ABB RAPID module: MainModule.mod

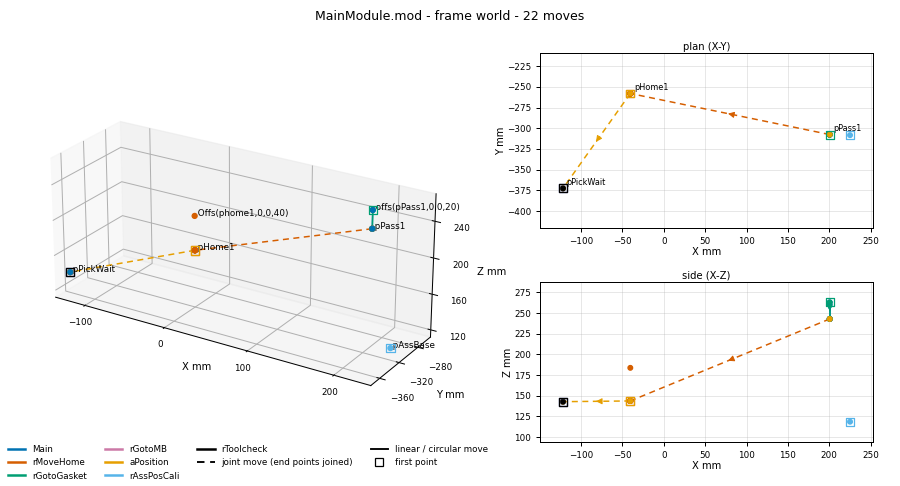
[picture p0: tool path of MainModule.mod in frame world, 22 of 155 moves have a stored position in this frame; points joined in program order, loops and branches not executed]
 MODULE MainModule
!*****************************************************
!Module Name: MainModule
!Version:     2.0
!Description: Menu Buttun and Gasket Assembly station
!Date:        2014\04\28
!Author:      Gavin Zhang
!*****************************************************
     PROC Main()
        VAR num X;
        VAR num Y;
        VAR string str_i;
        VAR pose poseCCD1;
        VAR pose poseTool;
        VAR num anglex;
        VAR num angley;
        VAR num anglez;
        rInitall;
        WHILE TRUE DO
            WHILE SocketStr<>"" DO
                IF SocketStr="robottest" THEN
                    FOR i FROM 1 TO 100 DO
                        SockGet:=FALSE;
                        MoveJ pPickWait,v200,z50,tGripper;
                        MoveL pCCD1,v200,fine,tGripper;
                        WaitTime 0.5;
                        SendStr:="ok";
                        SocketStr:="";
                        WaitUntil SendStr="";
                        waittime 0.5;
                        SockGet:=TRUE;
                        WaitUntil SocketStr="ok,ccd1check";
                        SocketStr:="";
                    ENDFOR
                    SockGet:=TRUE;
                ELSEIF SocketStr="robottest2" THEN
                    FOR i FROM 1 TO 50 DO
                        SockGet:=FALSE;
                        MoveL offs(pCCD1,0,0,20),v200,fine,tGripper;
                        MoveL pCCD1,v200,fine,tGripper;
                        MoveL offs(pCCD1,0,0,20),v200,fine,tGripper;
                        MoveJ offs(pPass1,0,0,20),v300,z10,tGripper;
                        MoveL pPass1,v600,z10,tGripper;
                        AccSet 50,50;
                        !MoveJ pInsert,v300,fine,tCurtool\WObj:=AssFrame;
                        MoveL pInsert,v300,fine,tCurtool\WObj:=AssFrame;
                        rInsert1;
                        WaitTime 0.5;
                        pActPos:=CRobT(\Tool:=tGripper\wobj:=wobj0);
                        MoveL offs(pActPos,0,0,20),v300,fine,tGripper\WObj:=wobj0;
                        MoveL offs(pCCD1,0,0,20),v200,fine,tGripper;
                        MoveL pCCD1,v200,fine,tGripper;
                        WaitTime 0.5;
                        SendStr:="ok";
                        SocketStr:="";
                        WaitUntil SendStr="";
                        waittime 0.5;
                        SockGet:=TRUE;
                        WaitUntil SocketStr="ok,ccd1check";
                        SocketStr:="";
                    ENDFOR
                    SockGet:=TRUE;
                ELSEIF SocketStr="ccd1check" THEN
                    SockGet:=FALSE;
                    !pCCD1Cali:=pCCD1;
                    MoveL pCCD1Cali,v100,fine,tGripper;
                    WaitTime\InPos,1;
                    SendStr:="ok,ccd1";
                    SocketStr:="";
                    WaitUntil SendStr="";
                    SockGet:=TRUE;
                    WaitUntil SocketStr="ok,ccd1";
                    SockGet:=FALSE;
                    pActPos:=CRobT(\Tool:=tGripper\wobj:=wobj0);
                    SendStr:="ok,"+ValToStr(pActPos.trans.X)+","+ValToStr(pActPos.trans.Y);
                    WaitUntil SendStr="";
                    SocketStr:="";
                    SockGet:=TRUE;
                    WaitUntil SocketStr="ccd1checkfinish";
                    SocketStr:="";
                    MoveJ pHome1,v100,fine,tGripper;
                    MoveJ pHome,v100,fine,tGripper;
                ELSEIF SocketStr="ccd2check" THEN
                    SockGet:=FALSE;
                    MoveJ phome,v100,z5,tGripper;
                    !MoveJ offs(pCCD2Cali,0,0,30),v100,z5,tGripper;
                    FOR i FROM 1 TO 9 DO
                        n:=trunc((i-1)/3);
                        b:=i-n*3;
                        pccd2Calib_T{i}:=offs(pCCD2Cali,(n-1)*2,(b-2)*2,0);
                    ENDFOR
                    FOR i FROM 1 TO 9 DO
                        MoveJ offs(pPickInkpad,0,0,140),v300,z5,tGripper;
                        MoveL pPickInkpad,v100,fine,tGripper;
                        WaitTime 0.5;
                        MoveL offs(pPickInkpad,0,0,140),v300,z5,tGripper;
                        SockGet:=FALSE;
                        MoveL offs(pccd2Calib_T{ARRAY{i}},0,0,30),v300,fine,tGripper;
                        MoveL pccd2Calib_T{ARRAY{i}},v100,fine,tGripper;
                        WaitTime\InPos,1;
                        pActPos:=CRobT(\Tool:=tGripper\wobj:=wobj0);
                        nPOSCCD2{i}:=pActPos.trans;
                        CCD2X{i}:=ValToStr(pActPos.trans.x);
                        CCD2y{i}:=ValToStr(pActPos.trans.y);
                        str_i:=ValToStr(i);
                        SendStr:="ok,"+str_i+","+CCD2X{i}+","+CCD2y{i};
                        WaitUntil SendStr="";
                        SocketStr:="";
                        SockGet:=TRUE;
                        IF i<>9 THEN
                            WaitUntil SocketStr="ok,ccd2";
                        ENDIF
                        WaitTime 1;
                        MoveL offs(pccd2Calib_T{ARRAY{i}},0,0,30),v300,fine,tGripper;
                    ENDFOR
                    SocketStr:="";
                    SockGet:=TRUE;
                    MoveJ phome,v100,z5,tGripper;
                ELSEIF SocketStr="gotomenubnt" THEN
                    SockGet:=FALSE;
                    rMoveHome;
                    MoveL pPickWait,v1000,fine,tGripper;
                    MoveL offs(pPick,0,0,30),v400,fine,tGripper;
                    MoveL pPick,v100,fine,tGripper;
                    SendStr:="ok";
                    SocketStr:="";
                    WaitUntil SendStr="";
                    SockGet:=TRUE;
                    !MoveL offs(pPick,0,0,30),v400,fine,tGripper;
                ELSEIF SocketStr="gotombccd" THEN
                    SockGet:=FALSE;
                    MoveL offs(pPick,0,0,30),v50,fine,tGripper;
                    !rMoveHome;
                    MoveL pCCD1,v600,fine,tGripper;
                    SendStr:="ok";
                    WaitTime 0.2;
                    SocketStr:="";
                    WaitUntil SendStr="";
                    SockGet:=TRUE;
                ELSEIF SocketStr="gotogasket" THEN
                    SockGet:=FALSE;
                    rMoveHome;
                    MoveJ pPass1,v600,z10,tCurTool;
                    MoveJ pInsert,v300,fine,tCurtool\WObj:=AssFrame;
                    !SocketSend socket1 \Str:="gotogasketfinish";
                    SendStr:="ok";
                    SocketStr:="";
                    WaitUntil SendStr="";
                    SockGet:=TRUE;
                ELSEIF SocketStr="gotoinitpos" THEN
                    SockGet:=FALSE;
                    rMoveHome;
                    !MoveJ pPass1,v600,z10,tGripper;
                    MoveJ pHome,v600,fine,tGripper;
                    SendStr:="ok";
                    SocketStr:="";
                    WaitUntil SendStr="";
                    SockGet:=TRUE;
                ELSEIF SocketStr="error" THEN
                    SockGet:=FALSE;
                    rMoveHome;
                    SendStr:="ok";
                    SocketStr:="";
                    WaitUntil SendStr="";
                    SockGet:=TRUE;
                ELSEIF SocketStr="startpress" THEN
                    SockGet:=FALSE;
                    rMoveHome;
                    MoveJ pPass1,v600,z10,tGripper;
                    rInsert1;
                    SendStr:="ok";
                    SocketStr:="";
                    WaitUntil SendStr="";
                    SockGet:=TRUE;
                ELSEIF SocketStr="calibtool" THEN
                    rTCPCalib1;
                ELSEIF SocketStr="ccd1calibration" THEN
                    rCCD1Calibration_1;
                ELSEIF SocketStr="calibtool5" THEN
                    rToolcheck;
                ELSEIF SocketStr="ccd2calibration" THEN
                    rCCD2Calibration;
                ELSEIF SocketStr="startwork" THEN
                    rWorkFlow;
                ELSEIF StrPart(SocketStr,1,15)="UpdateRobotData" THEN
                    tJogbycp;
                ENDIF
                rCyclecheck;
            ENDWHILE
            WaitTime 0.2;
        ENDWHILE
    ENDPROC

    PROC rInitall()
        WHILE diCalibration=1 DO
            TPErase;
            TPWrite "The Safe_Door is Opened,Please Close it";
            WaitDI diCalibration,0;
        ENDWHILE
        StartMove;
        AccSet 5,5;
        rMoveHome;
        bEmptyDone:=FALSE;
        SockGet:=TRUE;
        SocketStr:="";
        Reset doRobError1;
        Reset doRobError2;
        Reset doRobError3;
        Reset doRobError4;
        Reset doSocketError;
        Set doReady1;
        IDelete iInitall;
        CONNECT iInitall WITH tInitiall;
        ISignalDI diRobReset,1,iInitall;
        IDelete iInitall;
        CONNECT iInitall WITH tInitiall;
        ISignalDI diHomePos,1,iInitall;
        IDelete iSocketError;
        CONNECT iSocketError WITH tSocketerror;
        ISignalDO doSocketError,1,iSocketError;
        IDelete iEmptydone;
        CONNECT iEmptydone WITH tEmptyDone;
        ISignalDI diEmptydone,1,iEmptydone;
        IDelete intDoor;
        CONNECT intDoor WITH tSafetyDoor;
        ISignalDI diCalibration,1,intDoor;
    ENDPROC

    !rWorkFlow:the robot normal working flow;

    PROC rWorkFlow()
        VAR string str_i;
        !MoveJ pHome,v1000,fine,tGripper;
        WaitUntil SocketStr="startwork";
        SockGet:=FALSE;
        rGotoMB;
        SockGet:=TRUE;
        WaitUntil SocketStr="gotombccd";
        SockGet:=FALSE;
        rGotoMBCCD;
        SockGet:=TRUE;
        WaitUntil SocketStr<>"";
        WaitUntil StrPart(SocketStr,1,10)="workoffset";
        !Stop;
        SockGet:=FALSE;
        rDataOffset;
        SockGet:=TRUE;
        WaitUntil SocketStr<>"";
        WaitUntil StrPart(SocketStr,1,12)="robot_ponits";
        !Stop;
        SockGet:=FALSE;
        rCCD12Offset;
        SockGet:=TRUE;
        WaitUntil SocketStr="gotogasket";
        SockGet:=FALSE;
        rGotoGasket;
        SockGet:=TRUE;
        WaitUntil SocketStr<>"";
        WaitUntil StrPart(SocketStr,1,5)="guide";
        SockGet:=FALSE;
        rCCD3Guide;
        SockGet:=TRUE;
        WaitUntil SocketStr="startpress";
        SockGet:=FALSE;
        rMBPress;
        SockGet:=TRUE;
        WaitTime 0.5;
        !WaitUntil SocketStr= "gotoinitpos";
        SockGet:=FALSE;
        rGotoHome;
        SockGet:=TRUE;
    ENDPROC

    PROC rCyclecheck()
        WaitTime 0.1;
        !SocketStr:="";
    ENDPROC

    PROC rMoveHome()
        VelSet 100,500;
        IF bCurPos(pHome1,tGripper,10,10,10,wobj0) THEN
            MoveJ pHome1,v500,fine,tGripper;
            MoveL pHome,v500,fine,tGripper;
        ENDIF
        IF bCurPos(pHome,tGripper,10,10,10,wobj0) THEN
            MoveL pHome,v500,fine,tGripper;
        ENDIF
        IF bCurPos(pPick,tGripper,10,10,10,wobj0) THEN
            MoveJ offs(pPick,0,0,20),v500,fine,tGripper;
            MoveJ pHome,v500,fine,tGripper;
        ENDIF
        IF bCurPos(pCCD1Cali,tGripper,10,10,10,wobj0) THEN
            !MoveJ pPass1, v500, fine, tGripper;
            MoveJ pHome1,v500,Z10,tGripper;
            MoveL pHome,v500,fine,tGripper;
        ENDIF
        IF bCurPos(pCCD2Cali,tGripper,30,30,10,wobj0) THEN
            MoveJ Offs(pCCD2Cali,0,0,30),v100,fine,tGripper;
            MoveL Offs(phome1,0,0,40),v500,fine,tGripper;
            MoveL pHome,v500,fine,tGripper;
        ENDIF
        IF bCurPos(ppass1,tGripper,10,10,10,wobj0) THEN
            MoveJ pHome1,v500,Z10,tGripper;
            MoveJ pHome,v500,fine,tGripper;
        ENDIF
        IF bCurPos(pInsert,tCurTool,10,10,10,AssFrame) THEN
            MoveJ pPass1,v500,fine,tGripper;
            MoveJ pHome1,v500,fine,tGripper;
            MoveJ pHome,v500,fine,tGripper;
        ENDIF
        IF bCurrentPos(pHome,tGripper)=FALSE THEN
            ! If no known position is found, check if the robot is in a specified
            ! window and move him to the first position in the program
            pActPos:=CRobT(\Tool:=tGripper\WObj:=wobj0);
            IF (pPick.trans.x-5<pActPos.trans.x AND pActPos.trans.x<pCCD2Cali.trans.x+10) AND (-370<pActPos.trans.Y AND pActPos.trans.Y<0) AND pActPos.trans.z>pCCD2Cali.trans.z+20 THEN
                MoveL offs(pActPos,0,0,60),v300,z20,tGripper;
                MoveJ pHome1,v500,fine,tGripper;
                MoveL pHome,v500,fine,tGripper;
            ELSE
                WHILE OpMode()<>OP_MAN_PROG DO
                    TPErase;
                    TPWrite "Please switch robot to Manual mode";
                    !TPErase;
                    Stop;
                    MoveJ pHome,v300,z20,tGripper;
                ENDWHILE
            ENDIF
        ENDIF
        !MoveJ pWait,v300,z20,tTool\wobj:=WobTable;
        !MoveJ pHome,v300,z20,tGripper;
    ENDPROC

    PROC rGotoHome()
        !MoveL Offs(pAssembly,0,0,30),vAssembly,z10,tCurtool;
        pActPos:=CRobT(\Tool:=tCurTool\WObj:=AssFrame1);
        MoveL Offs(pActPos,0,0,5),v5,z1,tCurTool\WObj:=AssFrame1;
        MoveL Offs(pActPos,0,0,10),v50,z1,tCurTool\WObj:=AssFrame1;
        ConfL\On;
        AccSet 10,10;
        MoveJ pHome,v1000,fine,tGripper;
        !SocketSend socket1 \Str:="gotoinitposfinish";
        SendStr:="gotoinitposfinish";
        SocketStr:="";
        WaitUntil SendStr="";
    ENDPROC

    PROC rCCD1Calibration()
        VAR string str_i;
        !SockGet:=FALSE;
        MoveJ phome,v100,z5,tGripper;
        tGripper.tframe.trans.x:=0;
        tGripper.tframe.trans.y:=0;
        !position pCCD1Cali is define in the View's center of the CCD1
        pCCD1Cali:=pCCD1;
        MoveL pCCD1Cali,v100,fine,tGripper;
        !ConfL\Off;
        !rTCPCalib;
        FOR i FROM 1 TO 9 DO
            SockGet:=FALSE;
            n:=trunc((i-1)/3);
            b:=i-n*3;
            MoveJ RelTool(offs(pCCD1Cali,(n-1)*4,(b-2)*2.2,0),0,0,0\Rz:=180),v100,fine,tGripper;
            WaitTime\InPos,1;
            SendStr:="ok,180d";
            WaitUntil SendStr="";
            SocketStr:="";
            SockGet:=TRUE;
            WaitUntil SocketStr="ok,ccd1";
            WaitTime 1;
            SockGet:=FALSE;
            MoveJ offs(pCCD1Cali,(n-1)*4,(b-2)*2.2,0),v100,fine,tGripper;
            WaitTime\InPos,1;
            pActPos:=CRobT(\Tool:=tGripper\wobj:=wobj0);
            nPOSCCD1{i}:=pActPos.trans;
            CCD1X{i}:=ValToStr(pActPos.trans.x);
            CCD1y{i}:=ValToStr(pActPos.trans.y);
            str_i:=ValToStr(i);
            !SocketSend socket1 \Str:="ok"+str_i+","+CCD1X{i}+","+CCD1y{i};
            SendStr:="ok,"+str_i+","+CCD1X{i}+","+CCD1y{i};
            WaitUntil SendStr="";
            SocketStr:="";
            SockGet:=TRUE;
            IF i<>9 THEN
                WaitUntil SocketStr="ok,ccd1";
            ENDIF
            WaitTime 1;
        ENDFOR
        WaitUntil SendStr="";
        SockGet:=TRUE;
        SocketStr:="";
        MoveJ phome,v100,z5,tGripper;
    ENDPROC

    PROC rCCD1Calibration_1()
        VAR string str_i;
        !SockGet:=FALSE;
        MoveJ phome,v100,z5,tGripper;
        tGripper.tframe.trans.x:=0;
        tGripper.tframe.trans.y:=0;
        !position pCCD1Cali is define in the View's center of the CCD1
        pCCD1Cali:=pCCD1;
        MoveL pCCD1Cali,v100,fine,tGrip2;
        !ConfL\Off;
        !rTCPCalib;
        FOR i FROM 1 TO 9 DO
            SockGet:=FALSE;
            n:=trunc((i-1)/3);
            b:=i-n*3;
            MoveJ offs(pCCD1Cali,(n-1)*4,(b-2)*2.2,0),v100,fine,tGrip2;
            WaitTime\InPos,1;
            pActPos:=CRobT(\Tool:=tGrip2\wobj:=wobj0);
            nPOSCCD1{i}:=pActPos.trans;
            CCD1X{i}:=ValToStr(pActPos.trans.x);
            CCD1y{i}:=ValToStr(pActPos.trans.y);
            str_i:=ValToStr(i);
            !SocketSend socket1 \Str:="ok"+str_i+","+CCD1X{i}+","+CCD1y{i};
            SendStr:="ok,"+str_i+","+CCD1X{i}+","+CCD1y{i};
            WaitUntil SendStr="";
            SocketStr:="";
            SockGet:=TRUE;
            IF i<>9 THEN
                WaitUntil SocketStr="ok,ccd1";
            ENDIF
            WaitTime 1;
        ENDFOR
        WaitUntil SendStr="";
        SockGet:=TRUE;
        SocketStr:="";
        MoveJ phome,v100,z5,tGripper;
    ENDPROC

    PROC rCCD2Calibration()
        VAR string str_i;
        !SockGet:=FALSE;
        MoveJ phome,v100,z5,tGripper;
        FOR i FROM 1 TO 9 DO
            n:=trunc((i-1)/3);
            b:=i-n*3;
            pccd2Calib{i}:=offs(pCCD2Cali,(n-1)*4,(b-2)*4,0);
        ENDFOR

        FOR i FROM 1 TO 9 DO
            MoveJ offs(pPickInkpad,0,0,140),v300,z5,tGripper;
            MoveL pPickInkpad,v100,fine,tGripper;
            WaitTime 0.5;
            MoveL offs(pPickInkpad,0,0,140),v300,z5,tGripper;
            SockGet:=FALSE;
            MoveL offs(pccd2Calib{ARRAY{i}},0,0,30),v300,fine,tGripper;
            MoveL pccd2Calib{ARRAY{i}},v100,fine,tGripper;
            WaitTime\InPos,1;
            pActPos:=CRobT(\Tool:=tGripper\wobj:=wobj0);
            nPOSCCD2{i}:=pActPos.trans;
            CCD2X{i}:=ValToStr(pActPos.trans.x);
            CCD2y{i}:=ValToStr(pActPos.trans.y);
            str_i:=ValToStr(i);
            SendStr:="ok,"+str_i+","+CCD2X{i}+","+CCD2y{i};
            WaitUntil SendStr="";
            SocketStr:="";
            SockGet:=TRUE;
            IF i<>9 THEN
                WaitUntil SocketStr="ok,ccd2";
            ENDIF
            WaitTime 1;
            MoveL offs(pccd2Calib{ARRAY{i}},0,0,30),v300,fine,tGripper;
        ENDFOR
        SocketStr:="";
        SockGet:=TRUE;
        MoveJ phome,v100,z5,tGripper;
        RETURN ;
        MoveJ pCCD2Cali,v100,z5,tGripper;
    ENDPROC

    PROC rMBPress()
        ConfL\Off;
        nanglex:=0;
        nangley:=0;
        AssFrame1.uframe.rot:=AssFrame.uframe.rot*OrientZYX(90,0,0);
        AssFrame1.uframe.trans:=AssFrame.uframe.trans;
        IF OpMode()=OP_MAN_PROG STOP;
        AccSet 5,5;
        MoveL RelTool(Offs(pAssembly,noffsy,noffsx,4.2),0,0,0\Rx:=nanglex\Ry:=nangley\Rz:=0),vSlow,fine,tCurtool\WObj:=AssFrame1;
        MoveL RelTool(Offs(pAssembly,noffsy,noffsx,0),0,0,0\Rx:=nanglex\Ry:=nangley\Rz:=0),vSlowA,fine,tCurtool\WObj:=AssFrame1;
        WaitTime 0.3;
        MoveL RelTool(Offs(pAssembly,noffsy,noffsx,2),0,0,0\Rx:=nanglex\Ry:=nangley\Rz:=0),vSlowA,fine,tCurtool\WObj:=AssFrame1;
        WaitTime 0.2;
        SendStr:="pressfinish";
        SocketStr:="";
        WaitUntil SendStr="";
    ENDPROC

    PROC rCCD3Guide()
        nStrlength:=StrLen(SocketStr);
        nfind:=StrFind(SocketStr,1,",");
        ok:=StrToVal(StrPart(SocketStr,nfind+1,nStrLength-nfind),X3);
        SendStr:="recvguide";
        AccSet 50,50;
        X3:=0;
        MoveL Reltool(pInsert,nccd3offsx,0,x3+nccd3offs),v20,z10,tCurTool\WObj:=AssFrame;
        MoveL Offs(RelTool(pInsert,nccd3offsx,1,X3+nccd3offs),0,0,-40),v50,fine,tCurTool\WObj:=AssFrame;
        IF OpMode()=OP_MAN_PROG STOP;
        rInsert1;
        SocketStr:="";
        WaitUntil SendStr="";
    ENDPROC

    PROC rGotoGasket()
        MoveJ offs(pCCD1,0,0,100),v400,z50,tGripper;
        MoveJ offs(pPass1,0,0,20),v300,z10,tGripper;
        MoveL pPass1,v600,z10,tGripper;
        AccSet 50,50;
        MoveL pInsert,v200,fine,tCurTool\WObj:=AssFrame;
        IF OpMode()=OP_MAN_PROG STOP;
        WaitTime\InPos,1.5;
        SendStr:="gotogasketfinish";
        SocketStr:="";
        WaitUntil SendStr="";
    ENDPROC

    PROC rCCD12Offset()
        nStrlength:=StrLen(SocketStr);
        nFind:=0;
        FOR i FROM 1 TO 6 DO
            nfind:=StrFind(SocketStr,nFind+1,",");
            nArray{i}:=nFind;
        ENDFOR
        sCCD:=StrPart(SocketStr,1,nArray{1}-1);
        ok:=StrToVal(StrPart(SocketStr,nArray{1}+1,nArray{2}-nArray{1}-1),X1);
        ok:=StrToVal(StrPart(SocketStr,nArray{2}+1,nArray{3}-nArray{2}-1),Y1);
        ok:=StrToVal(StrPart(SocketStr,nArray{3}+1,nArray{4}-nArray{3}-1),nAngle1);
        ok:=StrToVal(StrPart(SocketStr,nArray{4}+1,nArray{5}-nArray{4}-1),X2);
        ok:=StrToVal(StrPart(SocketStr,nArray{5}+1,nArray{6}-nArray{5}-1),Y2);
        ok:=StrToVal(StrPart(SocketStr,nArray{6}+1,nStrLength-nArray{6}-1),nAngle2);
        SendStr:="recvok";
        rCalibTool X1,Y1,nAngle1;
        rDefAssFrame;
        WaitUntil SendStr="";
        SocketStr:="";
    ENDPROC

    PROC rDataOffset()
        nStrlength:=StrLen(SocketStr);
        nFind:=0;
        FOR i FROM 1 TO 6 DO
            nfind:=StrFind(SocketStr,nFind+1,",");
            nArray{i}:=nFind;
        ENDFOR
        sCCD:=StrPart(SocketStr,1,nArray{1}-1);
        ok:=StrToVal(StrPart(SocketStr,nArray{1}+1,nArray{2}-nArray{1}-1),noffsX);
        ok:=StrToVal(StrPart(SocketStr,nArray{2}+1,nArray{3}-nArray{2}-1),noffsY);
        ok:=StrToVal(StrPart(SocketStr,nArray{3}+1,nArray{4}-nArray{3}-1),noffsAngle);
        ok:=StrToVal(StrPart(SocketStr,nArray{4}+1,nArray{5}-nArray{4}-1),nAssX);
        ok:=StrToVal(StrPart(SocketStr,nArray{5}+1,nArray{6}-nArray{5}-1),nAssY);
        ok:=StrToVal(StrPart(SocketStr,nArray{6}+1,nStrLength-nArray{6}-1),nAssz);
        SendStr:="recvworkoffsetmsg";
        WaitUntil SendStr="";
        SocketStr:="";
    ENDPROC

    PROC rProcessFinish()
        rMoveHome;
        !SocketSend socket1 \Str:="resetmovefinish";
        SendStr:="resetmovefinish";
        WaitTime 0.2;
        SocketStr:="";
        WaitUntil SendStr="";
    ENDPROC

    PROC rGotoMBCCD()
        MoveL offs(pCCD1,0,0,60),v400,z100,tGripper;
        MoveL pCCD1,v200,fine,tGripper;
        WaitTime\InPos,0.5;
        SendStr:="gotombccdfinish";
        SocketStr:="";
        WaitUntil SendStr="";
    ENDPROC

    PROC rGotoMB()
        MoveL pHome,v1000,fine,tGripper;
        MoveL pPickWait,v1000,z200,tGripper;
        MoveL offs(pPick,0,0,5),v400,z10,tGripper;
        MoveL pPick,v20,fine,tGripper;
        SendStr:="gotomenubntfinish";
        WaitTime 0.5;
        MoveL offs(pPick,0,0,2.5),vSlow,fine,tGripper;
        MoveL offs(pPick,0,0,10),v400,z100,tGripper;
        SocketStr:="";
        WaitUntil SendStr="";
    ENDPROC

    !rInser:the insert action to assembly of the robot

    PROC rInsert1()
        nPoseAss:=[[-nAssy,nAssx,nAssz],[1,0,0,0]];
        PDispSet nPoseAss;
        MoveL p20,vAssembly,z1,tCurTool\WObj:=AssFrame;
        MoveL p30,vAssembly,z1,tCurTool\WObj:=AssFrame;
        MoveL p40,vAssembly,z1,tCurTool\WObj:=AssFrame;
        MoveL p50,vAssembly,z1,tCurTool\WObj:=AssFrame;
        MoveL p60,vAssembly,z1,tCurTool\WObj:=AssFrame;
        MoveL p70,vAssembly,z1,tCurTool\WObj:=AssFrame;
        MoveL p80,vAssembly,z1,tCurTool\WObj:=AssFrame;
        MoveL p90,vAssembly,z1,tCurTool\WObj:=AssFrame;
        MoveL p100,vAssembly,z1,tCurTool\WObj:=AssFrame;
        MoveL p110,vAssembly,z1,tCurTool\WObj:=AssFrame;
        MoveL p120,vAssembly,z1,tCurTool\WObj:=AssFrame;
        MoveL p130,vAssembly,z1,tCurTool\WObj:=AssFrame;
        MoveL p150,vAssembly,z1,tCurTool\WObj:=AssFrame;
        PDispOff;
        RETURN ;
        MoveL p180,vAssembly,z1,tGripper\WObj:=wobj0;
        MoveL p190,vAssembly,z1,tGripper\WObj:=wobj0;
        MoveL p200,vAssembly,z1,tGripper\WObj:=wobj0;
        MoveL p210,vAssembly,z1,tGripper\WObj:=wobj0;
        MoveL p220,vAssembly,z1,tGripper\WObj:=wobj0;
    ENDPROC

    PROC tJogbycp()
        nfind:=0;
        nTempX:=0;
        nTempY:=0;
        nTempZ:=0;
        nTAnglez:=0;
        nTAngley:=0;
        nTAnglex:=0;
        nPositionNo:=0;
        nHtemp:=0;
        FOR i FROM 1 TO 2 DO
            nfind:=StrFind(SocketStr,nFind+1,",");
            nArray1{i}:=nFind;
        ENDFOR
        sFirstStr:=StrPart(SocketStr,1,nArray1{1}-1);
        sSecondStr:=StrPart(SocketStr,nArray1{1}+1,nArray1{2}-nArray1{1}-1);
        IF sSecondStr="gotopoint" THEN
            nStrlength:=StrLen(SocketStr);
            nFind:=0;
            FOR i FROM 1 TO 3 DO
                nfind:=StrFind(SocketStr,nFind+1,",");
                nArray1{i}:=nFind;
            ENDFOR
            sFirstStr:=StrPart(SocketStr,1,nArray1{1}-1);
            sSecondStr:=StrPart(SocketStr,nArray1{1}+1,nArray1{2}-nArray1{1}-1);
            ok:=StrToVal(StrPart(SocketStr,nArray1{2}+1,nArray1{3}-nArray1{2}-1),nPositionNo);
            ok:=StrToVal(StrPart(SocketStr,nArray1{3}+1,nStrLength-nArray1{3}),nHtemp);
            TEST nPositionNo
            CASE 141:
                !141 Gasket Calibration position
                MoveL offs(pCCD2Cali,0,0,nHtemp),v50,fine,tGripper;
                !MoveL pCCD2Cali, v200, fine, tGripper;
            CASE 16:
                !Guide take picture position
                MoveL offs(pInsert,0,0,nHtemp),v50,fine,tCurtool\WObj:=AssFrame;
                !MoveL pInsert, v200, fine, tCurtool\WObj:=AssFrame;
            CASE 142:
                !Gasket calibration pick inkpad position
                MoveL offs(pPickInkpad,0,0,nHtemp),v50,fine,tGripper;
                !MoveL pPickInkpad, v200, fine, tGripper;
            CASE 350:
                !pick the menu buttun position
                MoveL offs(pPick,0,0,nHtemp),v50,fine,tGripper;
                !MoveL pPick, v200, fine, tGripper;
            CASE 351:
                !menu buttun calibration position
                MoveL offs(pCCD1,0,0,nHtemp),v50,fine,tGripper;
                !MoveL pCCD1, v200, fine, tGripper;
            CASE 352:
                !the home position
                MoveL offs(pHome,0,0,nHtemp),v50,fine,tGripper;
                !MoveL pHome, v200, fine, tGripper;
            ENDTEST
            SockGet:=FALSE;
            rBackVal;
            SockGet:=TRUE;
        ELSEIF sSecondStr="updatemove" THEN
            nStrlength:=StrLen(SocketStr);
            nFind:=0;
            FOR i FROM 1 TO 8 DO
                nfind:=StrFind(SocketStr,nFind+1,",");
                nArray1{i}:=nFind;
            ENDFOR
            sFirstStr:=StrPart(SocketStr,1,nArray1{1}-1);
            sSecondStr:=StrPart(SocketStr,nArray1{1}+1,nArray1{2}-nArray1{1}-1);
            sFrame:=StrPart(SocketStr,nArray1{2}+1,nArray1{3}-nArray1{2}-1);
            ok:=StrToVal(StrPart(SocketStr,nArray1{3}+1,nArray1{4}-nArray1{3}-1),nTempX);
            ok:=StrToVal(StrPart(SocketStr,nArray1{4}+1,nArray1{5}-nArray1{4}-1),nTempY);
            ok:=StrToVal(StrPart(SocketStr,nArray1{5}+1,nArray1{6}-nArray1{5}-1),nTempZ);
            ok:=StrToVal(StrPart(SocketStr,nArray1{6}+1,nArray1{7}-nArray1{6}-1),nTAnglez);
            ok:=StrToVal(StrPart(SocketStr,nArray1{7}+1,nArray1{8}-nArray1{7}-1),nTAngley);
            ok:=StrToVal(StrPart(SocketStr,nArray1{8}+1,nStrLength-nArray1{8}-1),nTAnglex);
            pActPos:=CRobT(\Tool:=tGripper\wobj:=wobj0);
            IF sFrame="tool" THEN
                MoveL RelTool(offs(pActPos,0,0,0),nTempX,nTempY,nTempZ\Rx:=-nTAnglex\Ry:=-nTAngley\Rz:=-nTAnglez),v50,fine,tGripper;
            ELSEIF sFrame="world" THEN
                MoveL RelTool(Offs(pActPos,nTempX,nTempY,nTempZ),0,0,0\Rx:=-nTAnglex\Ry:=-nTAngley\Rz:=-nTAnglez),v50,fine,tGripper;
            ENDIF
            SockGet:=FALSE;
            rBackVal;
            SockGet:=TRUE;
        ELSEIF sSecondStr="savepoint" THEN
            nStrlength:=StrLen(SocketStr);
            nFind:=0;
            FOR i FROM 1 TO 2 DO
                nfind:=StrFind(SocketStr,nFind+1,",");
                nArray1{i}:=nFind;
            ENDFOR
            sFirstStr:=StrPart(SocketStr,1,nArray1{1}-1);
            sSecondStr:=StrPart(SocketStr,nArray1{1}+1,nArray1{2}-nArray1{1}-1);
            ok:=StrToVal(StrPart(SocketStr,nArray1{2}+1,nStrLength-nArray1{2}),nPositionNo);
            TEST nPositionNo
            CASE 141:
                !141 Gasket Calibration position
                pActPos:=CRobT(\Tool:=tGripper\wobj:=wobj0);
                pCCD2Cali:=pActPos;
            CASE 16:
                !Guide take picture position
                pActPos:=CRobT(\Tool:=tCurtool\wobj:=AssFrame);
                pInsert:=pActPos;
            CASE 142:
                !Gasket calibration pick inkpad position
                pActPos:=CRobT(\Tool:=tGripper\wobj:=wobj0);
                pPickInkpad:=pActPos;
            CASE 350:
                !pick the menu buttun position
                pActPos:=CRobT(\Tool:=tGripper\wobj:=wobj0);
                pPick:=pActPos;
            CASE 351:
                !menu buttun calibration position
                pActPos:=CRobT(\Tool:=tGripper\wobj:=wobj0);
                pCCD1:=pActPos;
            CASE 352:
                !the home position
                pActPos:=CRobT(\Tool:=tGripper\wobj:=wobj0);
                pHome:=pActPos;
            ENDTEST
            SockGet:=FALSE;
            rBackVal;
            SockGet:=TRUE;
        ELSEIF sSecondStr="updatetool" THEN
            SockGet:=FALSE;
            WaitTime 0.5;
            SockGet:=TRUE;
        ELSEIF sSecondStr="updatehere" THEN
            SockGet:=FALSE;
            rBackVal;
            SockGet:=TRUE;
        ENDIF
        SockGet:=TRUE;
    ENDPROC

    PROC aPosition()
        MoveJ phome1,vAssembly,z1,tGripper;
        MoveJ pPickWait,vAssembly,z1,tGripper;
        MoveJ pCCD1Cali,vAssembly,z1,tGripper;
        MoveJ offs(pCCD2Cali,0,0,50),vAssembly,z1,tGripper;
        MoveJ pCCD2Cali,vAssembly,z1,tGripper;
        MoveJ offs(pCCD2Cali,0,0,50),vAssembly,z1,tGripper;
        MoveJ pCCD1,vAssembly,z1,tGripper;
        MoveJ pPickInkpad,vAssembly,z1,tGripper;
        MoveJ pPass1,vAssembly,z1,tGripper;
        MoveJ offs(pPick,0,0,50),vAssembly,z1,tGripper;
        MoveJ pPick,vAssembly,z1,tGripper;
        MoveJ offs(pPick,0,0,50),vAssembly,z1,tGripper;
        MoveL pInsert,vAssembly,z1,tcurtool\WObj:=AssFrame;
    ENDPROC

    PROC rCCD2Data(num n,robtarget pos)
        VAR string str_i;
        SockGet:=FALSE;
        MoveL offs(pos,0,0,10),v100,fine,tcp2;
        MoveL pos,v50,fine,tcp2;
        WaitTime 0.2;
        pActPos:=CRobT(\Tool:=tcp2\wobj:=wobj0);
        nPOSCCD1{n}:=pActPos.trans;
        CCD2X{n}:=ValToStr(pActPos.trans.x);
        CCD2y{n}:=ValToStr(pActPos.trans.y);
        str_i:=ValToStr(n);
        sendStr:="ok"+str_i+","+ccd2X{n}+","+ccd2y{n};
        WaitUntil SendStr="";
        SocketStr:="";
        SockGet:=TRUE;
        IF n<>9 THEN
            WaitUntil SocketStr="ok,ccd2";
        ENDIF
        MoveL offs(pos,0,0,10),v100,fine,tcp2;
    ENDPROC

    !the rCalibtool is Updata the tool of the robot
    PROC rCalibTool(
     num x,num y,num angle)
        VAR pose poseCCD1;
        VAR pose poseTool;
        VAR num anglex;
        VAR num angley;
        VAR num anglez;
        !MoveJ pCCD1, v500, fine, tGripper;
        !SocketGet sCCD1;
        !data from camera 1
        !CCD1_X: the X value of the feature point in the world coordinate
        posRel.trans.x:=X;
        posRel.trans.y:=Y;
        !posRel.trans.z := 108;
        posRel.trans.z:=pCCD1.trans.z;
        posRel.rot:=pCCD1.rot;
        anglez:=90+EulerZYX(\Z,pCCD1.rot);
        reg1:=anglez;
        !
        !nAngle:=anglez; ! delete for real test
        !posRel.rot := posRel.rot*OrientZYX(nAngle1-anglez,0,0);
        posRel.rot:=posRel.rot*OrientZYX(-Angle+90-noffsangle+anglez,0,0);
        !poseCCD1: pose where to take picture
        poseCCD1.trans:=pCCD1.trans;
        poseCCD1.rot:=pCCD1.rot;
        tCurTool:=tGripper;
        !calculate the actual tool data
        poseTool:=PoseMult(PoseInv(poseCCD1),posRel);
        poseTool:=PoseMult(tGripper.tframe,poseTool);
        !MoveJ pTemp, v1000, fine, tCurTool;
        !MoveJ reltool(pTemp,0,0,0\rz:=-180), v1000, fine, tCurTool;
        !poseTool.trans.z:=108;
        tCurtool.tframe.trans:=poseTool.trans;
        tCurtool.tframe.rot:=poseTool.rot;
    ENDPROC

    PROC rCalibTool1()
        VAR pose poseCCD1;
        VAR pose poseTool;
        VAR num anglex;
        VAR num angley;
        VAR num anglez;
        !MoveJ pCCD1, v500, fine, tGripper;
        !SocketGet sCCD1;
        !data from camera 1
        !CCD1_X: the X value of the feature point in the world coordinate
        posRel.trans.x:=X4;
        posRel.trans.y:=Y4;
        posRel.trans.z:=0;
        !posRel.trans.z := pCCD1.trans.z;
        posRel.rot:=pCCD1.rot;
        anglez:=EulerZYX(\Z,pCCD1.rot);
        reg1:=anglez;
        !
        !nAngle:=anglez; ! delete for real test
        posRel.rot:=posRel.rot*OrientZYX(nAngle4-anglez+180,0,0);
        !poseCCD1: pose where to take picture
        poseCCD1.trans:=pCCD1.trans;
        poseCCD1.rot:=pCCD1.rot;
        tCurTool:=tGripper;
        !calculate the actual tool data
        poseTool:=PoseMult(PoseInv(poseCCD1),posRel);
        poseTool.trans.z:=108;
        tCurtool.tframe.trans:=poseTool.trans;
        tCurtool.tframe.rot:=poseTool.rot;
    ENDPROC

    PROC rGripUpdata()
        VAR pose poseCCD1;
        VAR pose poseTool;
        VAR num anglex;
        VAR num angley;
        VAR num anglez;
        !SocketGet sCCD1;
        !data from camera 1
        !CCD1_X: the X value of the feature point in the world coordinate
        posRel.trans.x:=X1;
        posRel.trans.y:=Y1;
        posRel.trans.z:=78;
        posRel.rot:=pCCD1.rot;
        anglez:=EulerZYX(\Z,pCCD1.rot);
        !
        !nAngle:=anglez; ! delete for real test
        posRel.rot:=posRel.rot*OrientZYX(nAngle1-anglez,0,0);
        !poseCCD1: pose where to take picture
        poseCCD1.trans:=pCCD1.trans;
        poseCCD1.rot:=pCCD1.rot;
        tCurTool:=tGrip;
        !calculate the actual tool data
        poseTool:=PoseMult(PoseInv(poseCCD1),posRel);
        tCurtool.tframe.trans:=poseTool.trans;
        tGripper.tframe.rot:=tGripper.tframe.rot*OrientZYX(180,0,0);
    ENDPROC

    !rAssposCali:Auto Updata the press position of the robot by the CCD2
    PROC rAssPosCali()
        ! the data from CCD2
        pAssembly.trans.x:=X2;
        pAssembly.trans.y:=Y2;
        !the Z value is the robot position value.
        pAssembly.trans.z:=pAssBase.trans.z;
        pAssembly.rot:=OrientZYX(nAngle2,0,0);
        pAssembly.robconf:=pAssBase.robconf;
        RETURN ;
        MoveJ pAssBase,v100,fine,tGripper;
    ENDPROC

    !rDefassFrame:Auto Updata the assembly Frame of the assembly work object by the CCD2;
    PROC rDefAssFrame()
        AssFrame:=wobj0;
        ! the data from CCD2
        AssFrame.uframe.trans.x:=X2;
        AssFrame.uframe.trans.y:=Y2;
        !the Z value is Input by Munal
        AssFrame.uframe.trans.z:=7;
        AssFrame.uframe.rot:=wobj0.uframe.rot*OrientZYX(nAngle2-90,0,0);
    ENDPROC

    ! rTCPCalib:Calibration the TCP through the roution by the CCD data.
    PROC rTCPCalib()
        VAR num TCP_X;
        VAR num TCP_y;
        VAR string x;
        VAR string y;
        VAR pos pos1;
        pTCPCalib:=RelTool(pCCD1Cali,-3,-3,0);
        SockGet:=FALSE;
        MoveJ RelTool(pTCPCalib,0,0,0),v100,fine,tGripper;
        WaitTime 0.5;
        !pActPos:=CRobT(\Tool:=tGripper\wobj:=wobj0);
        !x:=ValToStr(pActPos.trans.x);
        !y:=ValToStr(pActPos.trans.y);
        SendStr:="ok,home";
        WaitUntil SendStr="";
        SocketStr:="";
        SockGet:=TRUE;
        WaitUntil SocketStr="ok,ccd1";
        MoveL RelTool(pTCPCalib,6,0,0),v100,fine,tGripper;
        WaitTime 0.5;
        SockGet:=FALSE;
        !SocketSend socket1 \Str:="x,6.0";
        SendStr:="ok,6.0";
        WaitUntil SendStr="";
        SocketStr:="";
        SockGet:=TRUE;
        WaitUntil SocketStr="ok,ccd1";
        MoveL pTCPCalib,v100,fine,tGripper;
        SockGet:=FALSE;
        MoveL RelTool(pTCPCalib,0,6,0),v100,fine,tGripper;
        WaitTime 0.5;
        SendStr:="ok,6.0";
        WaitUntil SendStr="";
        SocketStr:="";
        SockGet:=TRUE;
        WaitUntil SocketStr="ok,ccd1";
        MoveL pTCPCalib,v100,fine,tGripper;
        SockGet:=FALSE;
        !ConfL\Off;
        MoveJ RelTool(pTCPCalib,0,0,0\Rz:=180),v100,fine,tGripper;
        WaitTime 0.5;
        SendStr:="ok,180d";
        WaitUntil SendStr="";
        SocketStr:="";
        SockGet:=TRUE;
        MoveJ pTCPCalib,v100,fine,tGripper;
        WaitUntil SocketStr<>"";
        nStrlength:=StrLen(SocketStr);
        nfind:=0;
        FOR i FROM 1 TO 2 DO
            nfind:=StrFind(SocketStr,nFind+1,",");
            nArray1{i}:=nFind;
        ENDFOR
        sCCD:=StrPart(SocketStr,1,nArray1{1}-1);
        ok:=StrToVal(StrPart(SocketStr,nArray1{1}+1,nArray1{2}-nArray1{1}-1),TCP_X);
        ok:=StrToVal(StrPart(SocketStr,nArray1{2}+1,nStrLength-nArray{2}-1),TCP_Y);
        pos1.x:=-TCP_X;
        pos1.Y:=-TCP_Y;
        pos1.Z:=0;
        tGripper.tframe.trans:=PoseVect(tgripper.tframe,Pos1);
    ENDPROC

    PROC rToolcheck()
        VAR num tx;
        VAR num ty;
        SockGet:=FALSE;
        !pCCD1Cali:=pCCD1;
        MoveL pHome,v1000,fine,tGripper;
        MoveL pPickWait,v1000,z200,tGripper;
        MoveL offs(pPick,0,0,5),v400,z10,tGripper;
        MoveL pPick,v20,fine,tGripper;
        SendStr:="ok,calibtool5";
        SocketStr:="";
        WaitUntil SendStr="";
        SockGet:=TRUE;
        WaitUntil SocketStr="ok,calibtool5";
        MoveL offs(pCCD1,0,0,20),v400,z100,tGripper;
        MoveL pCCD1,v400,fine,tGripper;
        SockGet:=FALSE;
        WaitTime 1;
        SendStr:="ok,calibtool5";
        SocketStr:="";
        WaitUntil SendStr="";
        SockGet:=TRUE;
        WaitTime 1;
        WaitUntil SocketStr<>"";
        nStrlength:=StrLen(SocketStr);
        nfind:=0;
        FOR i FROM 1 TO 2 DO
            nfind:=StrFind(SocketStr,nFind+1,",");
            nArray1{i}:=nFind;
        ENDFOR
        sCCD:=StrPart(SocketStr,1,nArray1{1}-1);
        ok:=StrToVal(StrPart(SocketStr,nArray1{1}+1,nArray1{2}-nArray1{1}-1),tx);
        ok:=StrToVal(StrPart(SocketStr,nArray1{2}+1,nStrLength-nArray{2}-1),ty);
        rCalibTool tx,ty,0;
        pActPos:=CRobT(\Tool:=tCurtool\wobj:=wobj0);
        SockGet:=FALSE;
        MoveL RelTool(pActPos,0,0,0\Rz:=180),v100,fine,tCurTool;
        SendStr:="ok,180,"+ValToStr(pActPos.trans.X)+","+ValToStr(pActPos.trans.Y);
        SocketStr:="";
        WaitUntil SendStr="";
        SockGet:=TRUE;
        WaitTime 1;
        WaitUntil SocketStr="ok,rot180";
        MoveL pHome,v1000,fine,tGripper;
        SockGet:=FALSE;
        MoveL offs(pPick,0,0,5),v400,z10,tGripper;
        SendStr:="ok,calibtool5";
        SocketStr:="";
        WaitUntil SendStr="";
        SockGet:=TRUE;
        WaitTime 1;
        WaitUntil SocketStr="ok,calibtool5";
        MoveJ pHome,v100,fine,tGripper;
    ENDPROC

    PROC rTCPCalib1()
        VAR num TCP_X;
        VAR num TCP_y;
        VAR string x;
        VAR string y;
        VAR pos pos1;
        pTCPCalib:=RelTool(pCCD1Cali,-2,-2,0);
        SockGet:=FALSE;
        MoveJ RelTool(pTCPCalib,0,0,0),v100,fine,tGripper;
        WaitTime 0.5;
        SendStr:="ok,1,0,0";
        WaitUntil SendStr="";
        SocketStr:="";
        SockGet:=TRUE;
        WaitUntil SocketStr="ok,calibtool";
        MoveL RelTool(pTCPCalib,4,0,0),v100,fine,tGripper;
        WaitTime 0.5;
        SockGet:=FALSE;
        SendStr:="ok,2,4,0";
        WaitUntil SendStr="";
        SocketStr:="";
        SockGet:=TRUE;
        WaitUntil SocketStr="ok,calibtool";
        MoveL pTCPCalib,v100,fine,tGripper;
        SockGet:=FALSE;
        MoveL RelTool(pTCPCalib,0,4,0),v100,fine,tGripper;
        WaitTime 0.5;
        SendStr:="ok,3,0,4";
        WaitUntil SendStr="";
        SocketStr:="";
        SockGet:=TRUE;
        WaitUntil SocketStr="ok,calibtool";
        MoveL pTCPCalib,v100,fine,tGripper;
        SockGet:=FALSE;
        !ConfL\Off;
        MoveJ RelTool(pTCPCalib,0,0,0\Rz:=180),v100,fine,tGripper;
        WaitTime 0.5;
        SendStr:="ok,180d";
        WaitUntil SendStr="";
        SocketStr:="";
        SockGet:=TRUE;
        MoveJ pTCPCalib,v100,fine,tGripper;
        WaitUntil SocketStr<>"";
        nStrlength:=StrLen(SocketStr);
        nfind:=0;
        FOR i FROM 1 TO 2 DO
            nfind:=StrFind(SocketStr,nFind+1,",");
            nArray1{i}:=nFind;
        ENDFOR
        sCCD:=StrPart(SocketStr,1,nArray1{1}-1);
        ok:=StrToVal(StrPart(SocketStr,nArray1{1}+1,nArray1{2}-nArray1{1}-1),TCP_X);
        ok:=StrToVal(StrPart(SocketStr,nArray1{2}+1,nStrLength-nArray{2}-1),TCP_Y);
        pos1.x:=-TCP_X/2;
        pos1.Y:=-TCP_Y/2;
        pos1.Z:=0;
        tGrip2:=tGripper;
        tGrip2.tframe.trans:=PoseVect(tGripper.tframe,Pos1);
    ENDPROC

    TRAP tSocketError
        StopMove\Quick;
        Reset doSocketError;
        ExitCycle;
    ENDTRAP

    TRAP tInitiall
        StopMove\Quick;
        !bInitall:=TRUE;
        bEmptyDone:=FALSE;
        bCalibration:=FALSE;
        bWork:=FALSE;
        ExitCycle;
    ENDTRAP

    TRAP tEmptyDone
        StopMove\Quick;
        bEmptyDone:=TRUE;
        bInitall:=FALSE;
        bCalibration:=FALSE;
        bWork:=FALSE;
        SockGet:=FALSE;
        SendStr:="resetmovefinish";
        WaitTime 0.2;
        SocketStr:="";
        WaitUntil SendStr="";
        SockGet:=TRUE;
        ExitCycle;
    ENDTRAP

    PROC rBackVal()
        pActPos:=CRobT(\Tool:=tGripper\wobj:=wobj0);
        Zangle:=EulerZYX(\Z,pActPos.rot);
        Yangle:=EulerZYX(\Y,pActPos.rot);
        Xangle:=EulerZYX(\X,pActPos.rot);
        SendStr:="1,"+ValToStr(pActPos.trans.x)+","+ValToStr(pActPos.trans.y)+","+ValToStr(pActPos.trans.z)+","+ValToStr(Zangle)+","+ValToStr(Yangle)+","+ValToStr(Xangle);
        WaitUntil SendStr="";
        SocketStr:="";
    ENDPROC

    PROC test1()
        pAssembly.rot:=pAssembly.rot*orientZyx(0,180,180);
    ENDPROC

    TRAP tSafetyDoor
        StopMove\Quick;
        TPErase;
        TPWrite "The Safety door is opened,Please close it";
        WaitDI diCalibration,0;
        TPErase;
        StartMove;
    ENDTRAP

ENDMODULE
